// TwinCAT 3 PLC project PLCOpenInterface
// Title: TcPLCOpenWrapper
// Company: Loupe
// ProjectVersion: 0.0.1
// ProgramVersion: 3.1.4024.0
// libraries:
//   Tc2_Standard, * (Beckhoff Automation GmbH)
//   Tc2_System, * (Beckhoff Automation GmbH)
//   Tc3_Module, * (Beckhoff Automation GmbH)
// project tree:
//   PLCOpen/DUT/ PLCOpenCallInternal.TcDUT (not stored), PLCOpenCallState.TcTLEO (not stored), PLCOpenCommandInternal.TcDUT, PLCOpenStatusBase.TcTLEO
//   PLCOpen/Interfaces/ IPLCOpenBase.TcIO, IPLCOpenCall.TcIO (not stored), IPLCOpenCommand.TcIO (not stored), IPLCOpenGroup.TcIO (not stored)
//   PLCOpen/POU/ PLCOpenCall.TcPOU (not stored), PLCOpenCallGroup.TcPOU (not stored), PLCOpenCallGroupType.TcDUT (not stored), PLCOpenCommand.TcPOU (not stored), PLCOpenCommandGroup.TcPOU (not stored), PLCOpenNullRemote.TcPOU
//   / PlcTask.TcTTO (not stored)
//   POUs/ MAIN.TcPOU
// real-time tasks:
//   TASK PlcTask: cycle T#10ms, priority 20, ADS port 350

// ---- PLCOpen/DUT/PLCOpenCommandInternal.TcDUT
TYPE PLCOpenCommandInternal :
STRUCT
	_Execute : BOOL;
	_Trig : BOOL;
	_status : PLCOpenStatusBase;
	_remote : IPLCOpenCall;
	_nullRemote : PLCOpenNullRemote;
	_commandGroups : ARRAY[0..19] OF IPLCOpenGroup;
	_parameterReader : CopyPV;
END_STRUCT
END_TYPE

// ---- PLCOpen/DUT/PLCOpenStatusBase.TcTLEO
{attribute 'qualified_only'}
TYPE PLCOpenStatusBase :
(
	ERR_OK := 0,
	ERROR := 1,	
	ABORTED := 2,	
	ENABLED_WAITING := 65533,	
	NOT_ENABLED := 65534,	
	BUSY := 65535	
);
END_TYPE

// ---- PLCOpen/Interfaces/IPLCOpenBase.TcIO
INTERFACE IPLCOpenBase

PROPERTY Busy : BOOL
GET
END_GET
END_PROPERTY

PROPERTY ConsumeDone : Bool
GET
END_GET
END_PROPERTY

PROPERTY Done : BOOL
GET
END_GET
END_PROPERTY

PROPERTY Error : BOOL
GET
END_GET
END_PROPERTY

END_INTERFACE

// ---- PLCOpen/POU/PLCOpenNullRemote.TcPOU
FUNCTION_BLOCK PLCOpenNullRemote IMPLEMENTS  IPLCOpenCall

METHOD Aborted : BOOL
END_METHOD

METHOD Errored : BOOL
VAR_INPUT
	ID : INT;
END_VAR
END_METHOD

METHOD Finished : BOOL
END_METHOD

{warning 'add method implementation '}
METHOD Start : BOOL
VAR_INPUT
	Command	: IPLCOpenCommand;
END_VAR
//TODO
END_METHOD

END_FUNCTION_BLOCK

// ---- POUs/MAIN.TcPOU
PROGRAM MAIN
VAR
	call : PLCOpenCall;
	command : PLCOpenCommand;
END_VAR

END_PROGRAM
